FUNCTION_BLOCK FB_AirBlow
VAR_INPUT
	bExecute			: BOOL;
END_VAR
VAR_OUTPUT
	bDone				: BOOL;
	bBusy				: BOOL;
	bError				: BOOL;
	wErrorID			: BOOL;
END_VAR
VAR
	
	_exeRisingEdge		: R_TRIG;
	_exeFallingEdge		: F_TRIG;
	_step				: INT := 0;
END_VAR

_exeRisingEdge(CLK := bExecute);
_exeFallingEdge(CLK := bExecute);

IF _exeFallingEdge.Q THEN
	bDone := FALSE;	
END_IF

END_FUNCTION_BLOCK

(* stored: Version 1.1.0.1, ProductVersion 3.1.4024.10
   POU FB_AirBlow: Id {b1b50801-06ee-4f09-a7cc-e81d42471be1}, SpecialFunc None *)
